{attribute addProperty BoxType "EK1100-0000-0018"}
{attribute addProperty Id "Beckhoff_EL2xxxEK1122Beckhoff_EL2xxxEK1122_8D0C4044162A_0001_EL2002_0000_0000EL2002_B180A8D3405A_0002_EL2002_0000_0016EL2002_B180A8D3405A_0003_EL2002_0000_0017EL2002_B180A8D3405A_0004_EL2002_0000_0018EL2002_B180A8D3405A_0005_EL2004_0000_0000EL2004_E7E37CC2567A_0006_EL2004_0000_0016EL2004_E7E37CC2567A_0007_EL2004_0000_0017EL2004_E7E37CC2567A_0008_EL2004_0000_0018EL2004_E7E37CC2567A_0009_EL2008_0000_0016EL2008_04E0E56B8811A_0010_EL2008_0000_0017EL2008_04E0E56B8811A_0011_EL2008_0000_0018EL2008_04E0E56B8811A_0012_EL2014_0000_0016EL2014_3135F16014818.5A_0013_EL2014_0000_0017EL2014_3135F16014818.5A_0014_EL2022_0000_0016EL2022_B180A8D3405A_0015_EL2022_0000_0017EL2022_B180A8D3405A_0016_EL2022_0000_0018EL2022_B180A8D3405A_0017_EL2024_0000_0016EL2024_E7E37CC2567A_0018_EL2024_0000_0017EL2024_E7E37CC2567A_0019_EL2024_0000_0018EL2024_E7E37CC2567A_0020_EL2024_0000_0019EL2024_E7E37CC2567A_0021_EL2024_0010_0016EL2024_E7E37CC2567A_0022_EL2024_0010_0017EL2024_E7E37CC2567A_0023_EL2024_0010_0018EL2024_E7E37CC2567A_0024_EL2032_0000_0000EL2032_1D732299648A_0025_EL2032_0000_0016EL2032_1D732299648A_0026_EL2032_0000_0017EL2032_1D732299648A_0027_EL2032_0000_0018EL2032_1D732299648A_0028_EL2034_0000_0016EL2034_799515979612A_0029_EL2034_0000_0017EL2034_799515979612A_0030_EL2034_0000_0018EL2034_799515979612A_0031_EL2042_0000_0016EL2042_B180A8D3405A_0032_EL2042_0000_0017EL2042_B180A8D3405A_0033_EL2042_0000_0018EL2042_B180A8D3405A_0034_EL2044_0000_0016EL2044_3135F16014818.5A_0035_EL2084_0000_0016EL2084_E7E37CC2567A_0036_EL2084_0000_0017EL2084_E7E37CC2567A_0037_EL2084_0000_0018EL2084_E7E37CC2567A_0038_EL2088_0000_0016EL2088_04E0E56B8811A_0039_EL2088_0000_0017EL2088_04E0E56B8811A_0040_EL2088_0000_0018EL2088_04E0E56B8811A_0041_EL2124_0000_0016EL2124_E7E37CC2567A_0042_EL2124_0000_0017EL2124_E7E37CC2567A_0043_EL2124_0000_0018EL2124_E7E37CC2567A_0044_EL2202_0000_0000EL2202_B180A8D3405A_0045_EL2202_0000_0016EL2202_C9013BB5567A_0046_EL2202_0000_0017EL2202_C9013BB5567A_0047_EL2202_0000_0018EL2202_C9013BB5567A_0048_EL2202_0000_0019EL2202_C9013BB5567A_0049_EL2202_0100_0016EL2202_1ED54DF912015A_0050_EL2202_0100_0017EL2202_1ED54DF912015A_0051_EL2202_0100_0018EL2202_1ED54DF912015A_0052_EL2202_0100_0019EL2202_1ED54DF912015A_0053_EL2212_0000_0018EL2212_6ED00A9316020A_0054_EL2212_0000_0019EL2212_6ED00A9316020A_0055_EL2212_0000_0020EL2212_49077CE316020A_0056_EL2212_0000_0021EL2212_49077CE316020A_0057_EL2212_0000_0022EL2212_49077CE316020A_0058_EL2212_0000_0023EL2212_49077CE316020A_0059_EL2252_0000_0000EL2252_D83D30C214418A_0060_EL2252_0000_0016EL2252_1BB70CD317622A_0061_EL2252_0000_0017EL2252_8A6C7BB319224A_0062_EL2252_0000_0018EL2252_8A6C7BB319224A_0063_EL2252_0000_0019EL2252_8A6C7BB319224A_0064_EL2252_0000_0020EL2252_8A6C7BB319224A_0065_EL2258_0000_0016EL2258_9EFD418A5616702A_0066_EL2258_0000_0017EL2258_5305AE3B5560695A_0067_EL2262_0000_0000EL2262_CED6AB5C11214A_0068_EL2262_0000_0001EL2262_BE12C22013617A_0069_EL2262_0000_0002EL2262_A80E6C9A28035A_0070_EL2262_0000_0003EL2262_A80E6C9A28035A_0071_EL2262_0000_0004EL2262_CDC800E632040A_0072_EL2602_0000_0016EL2602_B180A8D3405A_0073_EL2602_0000_0017EL2602_B180A8D3405A_0074_EL2602_0000_0018EL2602_B180A8D3405A_0075_EL2602_0010_0016EL2602_0939F1F7567A_0076_EL2612_0000_0016EL2612_B180A8D3405A_0077_EL2612_0000_0017EL2612_B180A8D3405A_0078_EL2612_0000_0018EL2612_B180A8D3405A_0079_EL2622_0000_0016EL2622_B180A8D3405A_0080_EL2622_0000_0017EL2622_B180A8D3405A_0081_EL2622_0000_0018EL2622_B180A8D3405A_0082_EL2622_0010_0016EL2622_0939F1F7567A_0083_EL2624_0000_0016EL2624_E7E37CC2567A_0084_EL2624_0000_0017EL2624_E7E37CC2567A_0085_EL2624_0000_0018EL2624_E7E37CC2567A_0086_EL2634_0000_0016EL2634_E7E37CC2567A_0087_EL2634_0000_0017EL2634_E7E37CC2567A_0088_EL2642_0000_0016EL2642_A8D73BA720826A_0089_EL2652_0000_0016EL2652_B180A8D3405A_0090_EL2652_0000_0017EL2652_B180A8D3405A_0091_EL2652_0000_0018EL2652_B180A8D3405A_0092_EL2712_0000_0016EL2712_B180A8D3405A_0093_EL2712_0000_0017EL2712_B180A8D3405A_0094_EL2722_0000_0016EL2722_B180A8D3405A_0095_EL2722_0010_0016EL2722_B180A8D3405A_0096_EL2732_0000_0016EL2732_B180A8D3405A_0097_EL2784_0000_0016EL2784_E7E37CC2567A_0098_EL2788_0000_0016EL2788_04E0E56B8811A_0099_EL2794_0000_0016EL2794_E7E37CC2567A_0100_EL2798_0000_0016EL2798_04E0E56B8811A_0101_EL2798_0000_0017EL2798_04E0E56B8811A_0102_EL2798_0000_0018EL2798_04E0E56B8811A_0103_EL2808_0000_0016EL2808_04E0E56B8811A_0104_EL2808_0000_0017EL2808_04E0E56B8811A_0105_EL2808_0000_0018EL2808_04E0E56B8811A_0106_EL2809_0000_0016EL2809_5A2A5F2915219A_0107_EL2809_0000_0017EL2809_5A2A5F2915219A_0108_EL2809_0000_0018EL2809_5A2A5F2915219A_0109_EL2819_0000_0016EL2819_CAFBAEBC20826A_0110_EL2819_0000_0017EL2819_CAFBAEBC20826A_0111_EL2819_0000_0018EL2819_CAFBAEBC20826A_0112_EL2828_0000_0016EL2828_04E0E56B8811A_0113_EL2828_0000_0017EL2828_04E0E56B8811A_0114_EL2872_0000_0016EL2872_5A2A5F2915219A_0115_EL2872_0000_0017EL2872_5A2A5F2915219A_0116_EL2872_0000_0018EL2872_5A2A5F2915219A_0117_EL2872_0000_0019EL2872_5A2A5F2915219A_0118_EL2872_0010_0016EL2872_5A2A5F2915219A_0119_EL2872_0010_0017EL2872_5A2A5F2915219A_0120_EL2872_0010_0018EL2872_5A2A5F2915219A_0121_EL2872_0010_0019EL2872_5A2A5F2915219A_0122_EL2878_0005_0016EL2878_4C8AEF8F10413A_0123_EL2889_0000_0016EL2889_5A2A5F2915219A_0124_EL2889_0000_0017EL2889_5A2A5F2915219A_0125_EL2889_0000_0018EL2889_5A2A5F2915219A_0126_ELM2642_0000_0016ELM2642_D281BFF320826A_0127_ELM2644_0000_0016ELM2644_8836D28424030A_0128_ELM2742_0000_0016ELM2742_D281BFF320826A_0129_ELM2744_0000_0016ELM2744_8836D28424030"}
{attribute addProperty CRC "1766346312"}
{attribute addProperty SizeInBites "23916"}
{attribute addProperty SizeInBytes "2989.5"}
TYPE Beckhoff_EL2xxx_69484E48 EXTENDS EK1100_179A0949 :
STRUCT
	{attribute addProperty Name "Beckhoff_EL2xxxEK1122"}
	Beckhoff_EL2xxxEK1122 : Beckhoff_EL2xxxEK1122_8D0C4044;
	{attribute addProperty Name "A_0001_EL2002_0000_0000"}
	A_0001_EL2002_0000_0000 : EL2002_B180A8D3;
	{attribute addProperty Name "A_0002_EL2002_0000_0016"}
	A_0002_EL2002_0000_0016 : EL2002_B180A8D3;
	{attribute addProperty Name "A_0003_EL2002_0000_0017"}
	A_0003_EL2002_0000_0017 : EL2002_B180A8D3;
	{attribute addProperty Name "A_0004_EL2002_0000_0018"}
	A_0004_EL2002_0000_0018 : EL2002_B180A8D3;
	{attribute addProperty Name "A_0005_EL2004_0000_0000"}
	A_0005_EL2004_0000_0000 : EL2004_E7E37CC2;
	{attribute addProperty Name "A_0006_EL2004_0000_0016"}
	A_0006_EL2004_0000_0016 : EL2004_E7E37CC2;
	{attribute addProperty Name "A_0007_EL2004_0000_0017"}
	A_0007_EL2004_0000_0017 : EL2004_E7E37CC2;
	{attribute addProperty Name "A_0008_EL2004_0000_0018"}
	A_0008_EL2004_0000_0018 : EL2004_E7E37CC2;
	{attribute addProperty Name "A_0009_EL2008_0000_0016"}
	A_0009_EL2008_0000_0016 : EL2008_04E0E56B;
	{attribute addProperty Name "A_0010_EL2008_0000_0017"}
	A_0010_EL2008_0000_0017 : EL2008_04E0E56B;
	{attribute addProperty Name "A_0011_EL2008_0000_0018"}
	A_0011_EL2008_0000_0018 : EL2008_04E0E56B;
	{attribute addProperty Name "A_0012_EL2014_0000_0016"}
	A_0012_EL2014_0000_0016 : EL2014_3135F160;
	{attribute addProperty Name "A_0013_EL2014_0000_0017"}
	A_0013_EL2014_0000_0017 : EL2014_3135F160;
	{attribute addProperty Name "A_0014_EL2022_0000_0016"}
	A_0014_EL2022_0000_0016 : EL2022_B180A8D3;
	{attribute addProperty Name "A_0015_EL2022_0000_0017"}
	A_0015_EL2022_0000_0017 : EL2022_B180A8D3;
	{attribute addProperty Name "A_0016_EL2022_0000_0018"}
	A_0016_EL2022_0000_0018 : EL2022_B180A8D3;
	{attribute addProperty Name "A_0017_EL2024_0000_0016"}
	A_0017_EL2024_0000_0016 : EL2024_E7E37CC2;
	{attribute addProperty Name "A_0018_EL2024_0000_0017"}
	A_0018_EL2024_0000_0017 : EL2024_E7E37CC2;
	{attribute addProperty Name "A_0019_EL2024_0000_0018"}
	A_0019_EL2024_0000_0018 : EL2024_E7E37CC2;
	{attribute addProperty Name "A_0020_EL2024_0000_0019"}
	A_0020_EL2024_0000_0019 : EL2024_E7E37CC2;
	{attribute addProperty Name "A_0021_EL2024_0010_0016"}
	A_0021_EL2024_0010_0016 : EL2024_E7E37CC2;
	{attribute addProperty Name "A_0022_EL2024_0010_0017"}
	A_0022_EL2024_0010_0017 : EL2024_E7E37CC2;
	{attribute addProperty Name "A_0023_EL2024_0010_0018"}
	A_0023_EL2024_0010_0018 : EL2024_E7E37CC2;
	{attribute addProperty Name "A_0024_EL2032_0000_0000"}
	A_0024_EL2032_0000_0000 : EL2032_1D732299;
	{attribute addProperty Name "A_0025_EL2032_0000_0016"}
	A_0025_EL2032_0000_0016 : EL2032_1D732299;
	{attribute addProperty Name "A_0026_EL2032_0000_0017"}
	A_0026_EL2032_0000_0017 : EL2032_1D732299;
	{attribute addProperty Name "A_0027_EL2032_0000_0018"}
	A_0027_EL2032_0000_0018 : EL2032_1D732299;
	{attribute addProperty Name "A_0028_EL2034_0000_0016"}
	A_0028_EL2034_0000_0016 : EL2034_79951597;
	{attribute addProperty Name "A_0029_EL2034_0000_0017"}
	A_0029_EL2034_0000_0017 : EL2034_79951597;
	{attribute addProperty Name "A_0030_EL2034_0000_0018"}
	A_0030_EL2034_0000_0018 : EL2034_79951597;
	{attribute addProperty Name "A_0031_EL2042_0000_0016"}
	A_0031_EL2042_0000_0016 : EL2042_B180A8D3;
	{attribute addProperty Name "A_0032_EL2042_0000_0017"}
	A_0032_EL2042_0000_0017 : EL2042_B180A8D3;
	{attribute addProperty Name "A_0033_EL2042_0000_0018"}
	A_0033_EL2042_0000_0018 : EL2042_B180A8D3;
	{attribute addProperty Name "A_0034_EL2044_0000_0016"}
	A_0034_EL2044_0000_0016 : EL2044_3135F160;
	{attribute addProperty Name "A_0035_EL2084_0000_0016"}
	A_0035_EL2084_0000_0016 : EL2084_E7E37CC2;
	{attribute addProperty Name "A_0036_EL2084_0000_0017"}
	A_0036_EL2084_0000_0017 : EL2084_E7E37CC2;
	{attribute addProperty Name "A_0037_EL2084_0000_0018"}
	A_0037_EL2084_0000_0018 : EL2084_E7E37CC2;
	{attribute addProperty Name "A_0038_EL2088_0000_0016"}
	A_0038_EL2088_0000_0016 : EL2088_04E0E56B;
	{attribute addProperty Name "A_0039_EL2088_0000_0017"}
	A_0039_EL2088_0000_0017 : EL2088_04E0E56B;
	{attribute addProperty Name "A_0040_EL2088_0000_0018"}
	A_0040_EL2088_0000_0018 : EL2088_04E0E56B;
	{attribute addProperty Name "A_0041_EL2124_0000_0016"}
	A_0041_EL2124_0000_0016 : EL2124_E7E37CC2;
	{attribute addProperty Name "A_0042_EL2124_0000_0017"}
	A_0042_EL2124_0000_0017 : EL2124_E7E37CC2;
	{attribute addProperty Name "A_0043_EL2124_0000_0018"}
	A_0043_EL2124_0000_0018 : EL2124_E7E37CC2;
	{attribute addProperty Name "A_0044_EL2202_0000_0000"}
	A_0044_EL2202_0000_0000 : EL2202_B180A8D3;
	{attribute addProperty Name "A_0045_EL2202_0000_0016"}
	A_0045_EL2202_0000_0016 : EL2202_C9013BB5;
	{attribute addProperty Name "A_0046_EL2202_0000_0017"}
	A_0046_EL2202_0000_0017 : EL2202_C9013BB5;
	{attribute addProperty Name "A_0047_EL2202_0000_0018"}
	A_0047_EL2202_0000_0018 : EL2202_C9013BB5;
	{attribute addProperty Name "A_0048_EL2202_0000_0019"}
	A_0048_EL2202_0000_0019 : EL2202_C9013BB5;
	{attribute addProperty Name "A_0049_EL2202_0100_0016"}
	A_0049_EL2202_0100_0016 : EL2202_1ED54DF9;
	{attribute addProperty Name "A_0050_EL2202_0100_0017"}
	A_0050_EL2202_0100_0017 : EL2202_1ED54DF9;
	{attribute addProperty Name "A_0051_EL2202_0100_0018"}
	A_0051_EL2202_0100_0018 : EL2202_1ED54DF9;
	{attribute addProperty Name "A_0052_EL2202_0100_0019"}
	A_0052_EL2202_0100_0019 : EL2202_1ED54DF9;
	{attribute addProperty Name "A_0053_EL2212_0000_0018"}
	A_0053_EL2212_0000_0018 : EL2212_6ED00A93;
	{attribute addProperty Name "A_0054_EL2212_0000_0019"}
	A_0054_EL2212_0000_0019 : EL2212_6ED00A93;
	{attribute addProperty Name "A_0055_EL2212_0000_0020"}
	A_0055_EL2212_0000_0020 : EL2212_49077CE3;
	{attribute addProperty Name "A_0056_EL2212_0000_0021"}
	A_0056_EL2212_0000_0021 : EL2212_49077CE3;
	{attribute addProperty Name "A_0057_EL2212_0000_0022"}
	A_0057_EL2212_0000_0022 : EL2212_49077CE3;
	{attribute addProperty Name "A_0058_EL2212_0000_0023"}
	A_0058_EL2212_0000_0023 : EL2212_49077CE3;
	{attribute addProperty Name "A_0059_EL2252_0000_0000"}
	A_0059_EL2252_0000_0000 : EL2252_D83D30C2;
	{attribute addProperty Name "A_0060_EL2252_0000_0016"}
	A_0060_EL2252_0000_0016 : EL2252_1BB70CD3;
	{attribute addProperty Name "A_0061_EL2252_0000_0017"}
	A_0061_EL2252_0000_0017 : EL2252_8A6C7BB3;
	{attribute addProperty Name "A_0062_EL2252_0000_0018"}
	A_0062_EL2252_0000_0018 : EL2252_8A6C7BB3;
	{attribute addProperty Name "A_0063_EL2252_0000_0019"}
	A_0063_EL2252_0000_0019 : EL2252_8A6C7BB3;
	{attribute addProperty Name "A_0064_EL2252_0000_0020"}
	A_0064_EL2252_0000_0020 : EL2252_8A6C7BB3;
	{attribute addProperty Name "A_0065_EL2258_0000_0016"}
	A_0065_EL2258_0000_0016 : EL2258_9EFD418A;
	{attribute addProperty Name "A_0066_EL2258_0000_0017"}
	A_0066_EL2258_0000_0017 : EL2258_5305AE3B;
	{attribute addProperty Name "A_0067_EL2262_0000_0000"}
	A_0067_EL2262_0000_0000 : EL2262_CED6AB5C;
	{attribute addProperty Name "A_0068_EL2262_0000_0001"}
	A_0068_EL2262_0000_0001 : EL2262_BE12C220;
	{attribute addProperty Name "A_0069_EL2262_0000_0002"}
	A_0069_EL2262_0000_0002 : EL2262_A80E6C9A;
	{attribute addProperty Name "A_0070_EL2262_0000_0003"}
	A_0070_EL2262_0000_0003 : EL2262_A80E6C9A;
	{attribute addProperty Name "A_0071_EL2262_0000_0004"}
	A_0071_EL2262_0000_0004 : EL2262_CDC800E6;
	{attribute addProperty Name "A_0072_EL2602_0000_0016"}
	A_0072_EL2602_0000_0016 : EL2602_B180A8D3;
	{attribute addProperty Name "A_0073_EL2602_0000_0017"}
	A_0073_EL2602_0000_0017 : EL2602_B180A8D3;
	{attribute addProperty Name "A_0074_EL2602_0000_0018"}
	A_0074_EL2602_0000_0018 : EL2602_B180A8D3;
	{attribute addProperty Name "A_0075_EL2602_0010_0016"}
	A_0075_EL2602_0010_0016 : EL2602_0939F1F7;
	{attribute addProperty Name "A_0076_EL2612_0000_0016"}
	A_0076_EL2612_0000_0016 : EL2612_B180A8D3;
	{attribute addProperty Name "A_0077_EL2612_0000_0017"}
	A_0077_EL2612_0000_0017 : EL2612_B180A8D3;
	{attribute addProperty Name "A_0078_EL2612_0000_0018"}
	A_0078_EL2612_0000_0018 : EL2612_B180A8D3;
	{attribute addProperty Name "A_0079_EL2622_0000_0016"}
	A_0079_EL2622_0000_0016 : EL2622_B180A8D3;
	{attribute addProperty Name "A_0080_EL2622_0000_0017"}
	A_0080_EL2622_0000_0017 : EL2622_B180A8D3;
	{attribute addProperty Name "A_0081_EL2622_0000_0018"}
	A_0081_EL2622_0000_0018 : EL2622_B180A8D3;
	{attribute addProperty Name "A_0082_EL2622_0010_0016"}
	A_0082_EL2622_0010_0016 : EL2622_0939F1F7;
	{attribute addProperty Name "A_0083_EL2624_0000_0016"}
	A_0083_EL2624_0000_0016 : EL2624_E7E37CC2;
	{attribute addProperty Name "A_0084_EL2624_0000_0017"}
	A_0084_EL2624_0000_0017 : EL2624_E7E37CC2;
	{attribute addProperty Name "A_0085_EL2624_0000_0018"}
	A_0085_EL2624_0000_0018 : EL2624_E7E37CC2;
	{attribute addProperty Name "A_0086_EL2634_0000_0016"}
	A_0086_EL2634_0000_0016 : EL2634_E7E37CC2;
	{attribute addProperty Name "A_0087_EL2634_0000_0017"}
	A_0087_EL2634_0000_0017 : EL2634_E7E37CC2;
	{attribute addProperty Name "A_0088_EL2642_0000_0016"}
	A_0088_EL2642_0000_0016 : EL2642_A8D73BA7;
	{attribute addProperty Name "A_0089_EL2652_0000_0016"}
	A_0089_EL2652_0000_0016 : EL2652_B180A8D3;
	{attribute addProperty Name "A_0090_EL2652_0000_0017"}
	A_0090_EL2652_0000_0017 : EL2652_B180A8D3;
	{attribute addProperty Name "A_0091_EL2652_0000_0018"}
	A_0091_EL2652_0000_0018 : EL2652_B180A8D3;
	{attribute addProperty Name "A_0092_EL2712_0000_0016"}
	A_0092_EL2712_0000_0016 : EL2712_B180A8D3;
	{attribute addProperty Name "A_0093_EL2712_0000_0017"}
	A_0093_EL2712_0000_0017 : EL2712_B180A8D3;
	{attribute addProperty Name "A_0094_EL2722_0000_0016"}
	A_0094_EL2722_0000_0016 : EL2722_B180A8D3;
	{attribute addProperty Name "A_0095_EL2722_0010_0016"}
	A_0095_EL2722_0010_0016 : EL2722_B180A8D3;
	{attribute addProperty Name "A_0096_EL2732_0000_0016"}
	A_0096_EL2732_0000_0016 : EL2732_B180A8D3;
	{attribute addProperty Name "A_0097_EL2784_0000_0016"}
	A_0097_EL2784_0000_0016 : EL2784_E7E37CC2;
	{attribute addProperty Name "A_0098_EL2788_0000_0016"}
	A_0098_EL2788_0000_0016 : EL2788_04E0E56B;
	{attribute addProperty Name "A_0099_EL2794_0000_0016"}
	A_0099_EL2794_0000_0016 : EL2794_E7E37CC2;
	{attribute addProperty Name "A_0100_EL2798_0000_0016"}
	A_0100_EL2798_0000_0016 : EL2798_04E0E56B;
	{attribute addProperty Name "A_0101_EL2798_0000_0017"}
	A_0101_EL2798_0000_0017 : EL2798_04E0E56B;
	{attribute addProperty Name "A_0102_EL2798_0000_0018"}
	A_0102_EL2798_0000_0018 : EL2798_04E0E56B;
	{attribute addProperty Name "A_0103_EL2808_0000_0016"}
	A_0103_EL2808_0000_0016 : EL2808_04E0E56B;
	{attribute addProperty Name "A_0104_EL2808_0000_0017"}
	A_0104_EL2808_0000_0017 : EL2808_04E0E56B;
	{attribute addProperty Name "A_0105_EL2808_0000_0018"}
	A_0105_EL2808_0000_0018 : EL2808_04E0E56B;
	{attribute addProperty Name "A_0106_EL2809_0000_0016"}
	A_0106_EL2809_0000_0016 : EL2809_5A2A5F29;
	{attribute addProperty Name "A_0107_EL2809_0000_0017"}
	A_0107_EL2809_0000_0017 : EL2809_5A2A5F29;
	{attribute addProperty Name "A_0108_EL2809_0000_0018"}
	A_0108_EL2809_0000_0018 : EL2809_5A2A5F29;
	{attribute addProperty Name "A_0109_EL2819_0000_0016"}
	A_0109_EL2819_0000_0016 : EL2819_CAFBAEBC;
	{attribute addProperty Name "A_0110_EL2819_0000_0017"}
	A_0110_EL2819_0000_0017 : EL2819_CAFBAEBC;
	{attribute addProperty Name "A_0111_EL2819_0000_0018"}
	A_0111_EL2819_0000_0018 : EL2819_CAFBAEBC;
	{attribute addProperty Name "A_0112_EL2828_0000_0016"}
	A_0112_EL2828_0000_0016 : EL2828_04E0E56B;
	{attribute addProperty Name "A_0113_EL2828_0000_0017"}
	A_0113_EL2828_0000_0017 : EL2828_04E0E56B;
	{attribute addProperty Name "A_0114_EL2872_0000_0016"}
	A_0114_EL2872_0000_0016 : EL2872_5A2A5F29;
	{attribute addProperty Name "A_0115_EL2872_0000_0017"}
	A_0115_EL2872_0000_0017 : EL2872_5A2A5F29;
	{attribute addProperty Name "A_0116_EL2872_0000_0018"}
	A_0116_EL2872_0000_0018 : EL2872_5A2A5F29;
	{attribute addProperty Name "A_0117_EL2872_0000_0019"}
	A_0117_EL2872_0000_0019 : EL2872_5A2A5F29;
	{attribute addProperty Name "A_0118_EL2872_0010_0016"}
	A_0118_EL2872_0010_0016 : EL2872_5A2A5F29;
	{attribute addProperty Name "A_0119_EL2872_0010_0017"}
	A_0119_EL2872_0010_0017 : EL2872_5A2A5F29;
	{attribute addProperty Name "A_0120_EL2872_0010_0018"}
	A_0120_EL2872_0010_0018 : EL2872_5A2A5F29;
	{attribute addProperty Name "A_0121_EL2872_0010_0019"}
	A_0121_EL2872_0010_0019 : EL2872_5A2A5F29;
	{attribute addProperty Name "A_0122_EL2878_0005_0016"}
	A_0122_EL2878_0005_0016 : EL2878_4C8AEF8F;
	{attribute addProperty Name "A_0123_EL2889_0000_0016"}
	A_0123_EL2889_0000_0016 : EL2889_5A2A5F29;
	{attribute addProperty Name "A_0124_EL2889_0000_0017"}
	A_0124_EL2889_0000_0017 : EL2889_5A2A5F29;
	{attribute addProperty Name "A_0125_EL2889_0000_0018"}
	A_0125_EL2889_0000_0018 : EL2889_5A2A5F29;
	{attribute addProperty Name "A_0126_ELM2642_0000_0016"}
	A_0126_ELM2642_0000_0016 : ELM2642_D281BFF3;
	{attribute addProperty Name "A_0127_ELM2644_0000_0016"}
	A_0127_ELM2644_0000_0016 : ELM2644_8836D284;
	{attribute addProperty Name "A_0128_ELM2742_0000_0016"}
	A_0128_ELM2742_0000_0016 : ELM2742_D281BFF3;
	{attribute addProperty Name "A_0129_ELM2744_0000_0016"}
	A_0129_ELM2744_0000_0016 : ELM2744_8836D284;
END_STRUCT
END_TYPE

(* stored: Version 1.2.0.0, ProductVersion 3.1.4024.9
   DUT Beckhoff_EL2xxx_69484E48: Id {7c36e7e0-bc6c-46fc-bfe3-9f7d3240d5c5} *)
